PROGRAM motionChalleng_moveAbs
VAR
    myAxis : AXIS_REF;
    mcPower : MC_Power;
    mcMoveAbs : MC_MoveAbsolute;
    highLimitPosition : LREAL := 500;
    lowLimitPosition : LREAL := -5;
    enableAxis : BOOL;
    
    userSetPoint : LREAL;
    defaultVelocity : LREAL := 50;
    executeMoveAbs : BOOL;
END_VAR

mcPower(Axis:= myAxis, Enable_Positive:= highLimit, Enable_Negative:= lowLimit, Enable:= enableAxis);

mcMoveAbs(Axis:= myAxis, Execute:= executeMoveAbs, Position:= userSetPoint, Velocity:= defaultVelocity);
IF mcMoveAbs.Done THEN
    executeMoveAbs:= FALSE;
END_IF

TRANSITION highLimit:
highLimit:= myAxis.NcToPlc.ActPos<highLimitPosition;
END_TRANSITION

TRANSITION lowLimit:
lowLimit:= myAxis.NcToPlc.ActPos>lowLimitPosition;
END_TRANSITION

END_PROGRAM

(* stored: Version 1.1.0.1, ProductVersion 3.1.4024.5
   POU motionChalleng_moveAbs: Id {2f9ff8db-892a-43f5-9876-798d3644c9ec}, SpecialFunc None
   Transition highLimit: Id {2ff71a4c-3b15-454a-b600-e6e17ba803c3}
   Transition lowLimit: Id {58585069-4e4a-4f69-9ade-489021734355} *)
